TEXTLIST FadeRate
  0 = 'Unknown'
  1 = '358 steps/s'
  2 = '253 steps/s'
  3 = '179 steps/s'
  4 = '127 steps/s'
  5 = '89,4 steps/s'
  6 = '63,3 steps/s'
  7 = '44,7 steps/s'
  8 = '31,6 steps/s'
  9 = '22,4 steps/s'
  10 = '15,8 steps/s'
  11 = '11,2 steps/s'
  12 = '7,9 steps/s'
  13 = '5,6 steps/s'
  14 = '4,0 steps/s'
  15 = '2,8 steps/s'
  255 = 'Unknown'
   = ''
END_TEXTLIST

(* stored: Version 1.1.0.1, ProductVersion 3.1.4024.12
   TextList FadeRate: Id {1a19d742-528a-4af2-b1fb-061cff25bac8} *)
